PROGRAM MAIN
VAR
END_VAR

// Test only purpose
// if the project is changed to library #remove this

END_PROGRAM

(* stored: Version 1.1.0.1, ProductVersion 3.1.4024.9
   POU MAIN: Id {28360960-9ab2-43c1-b11c-05f0dfab6dbb}, SpecialFunc None *)
